// TIA Portal V18 export
DATA_BLOCK "KistlerPresser1_DB"   // DB2312
{ S7_Optimized_Access := 'FALSE' }
// stored: AutoNumber false
   VAR
      ShaftID : Array[0..50] of Char;
      HousingID_1 : Array[0..50] of Char;
      HousingID_2 : Array[0..50] of Char;
      Shaft : String[48];
      spare : String[48] := '46';
   END_VAR
BEGIN
END_DATA_BLOCK
